(* PLC project binary_encoder, Dassault Systèmes ControlBuild 2024x *)
(* stored: creationDateTime 2023-10-03T11:12:52-01:00 *)

(* This module simulates the behaviour of a binary encoder *)
FUNCTION_BLOCK equipment_library.binary_encoder
  VAR_INPUT
    binaryInput : DINT := 0;
    encoderFreezing : BOOL := false;
  END_VAR
  VAR_OUTPUT
    bit00 : BOOL := false;
    bit01 : BOOL := false;
    bit02 : BOOL := false;
    bit03 : BOOL := false;
    bit04 : BOOL := false;
    bit05 : BOOL := false;
    bit06 : BOOL := false;
    bit07 : BOOL := false;
    bit08 : BOOL := false;
    bit09 : BOOL := false;
    bit10 : BOOL := false;
    bit11 : BOOL := false;
    bit12 : BOOL := false;
    bit13 : BOOL := false;
    bit14 : BOOL := false;
    bit15 : BOOL := false;
    bit16 : BOOL := false;
    wordOutput : DINT := 0;
  END_VAR
  VAR
    inputValue : DINT := 0;
    parity : BOOL := false;
  END_VAR
  VAR CONSTANT
    evenParity : BOOL := false;
    oddParity : BOOL := true;
  END_VAR
  VAR
    d_presetting : BOOL := false;
    v_d_presetting : DINT := 0;
  END_VAR


ACTION C_source_code:
/* ----------------------------------------------------------------	*/
/* Type : Model of Operative Behaviour					*/
/* Category :  Sensors							*/
/* Author : Dassault Systemes						*/
/* Update date : June 2018							*/
/* ----------------------------------------------------------------	*/
/* This module simulates the behaviour 					*/
/* of a binary encoder.							*/
/* The whole value is encoded on 15 bits					*/
/*	the 16th bit is the parity bit. 					*/
/* ----------------------------------------------------------------	*/

/* ----------------------------------------------------------------	*/
/* Treatment of presetting fault						*/
/* ----------------------------------------------------------------	*/
if (d_presetting) inputValue = v_d_presetting;
else inputValue = binaryInput;


/* ----------------------------------------------------------------	*/
/* Encoder management							*/
/* ----------------------------------------------------------------	*/
if (!encoderFreezing) {
	bit00 = 0;
	bit01 = 0;
	bit02 = 0;
	bit03 = 0;
	bit04 = 0;
	bit05 = 0;
	bit06 = 0;
	bit07 = 0;
	bit08 = 0;
	bit09 = 0;
	bit10 = 0;
	bit11 = 0;
	bit12 = 0;
	bit13 = 0;
	bit14 = 0;
	bit15 = 0;

	if ((inputValue & 1)>0) bit00 = 1;
	if ((inputValue & 2)>0) bit01 = 1;
	if ((inputValue & 4)>0) bit02 = 1;
	if ((inputValue & 8)>0) bit03 = 1;
	if ((inputValue & 16)>0) bit04 = 1;
	if ((inputValue & 32)>0) bit05 = 1;
	if ((inputValue & 64)>0) bit06 = 1;
	if ((inputValue & 128)>0) bit07 = 1;
	if ((inputValue & 256)>0) bit08 = 1;
	if ((inputValue & 512)>0) bit09 = 1;
	if ((inputValue & 1024)>0) bit10 = 1;
	if ((inputValue & 2048)>0) bit11 = 1;
	if ((inputValue & 4096)>0) bit12 = 1;
	if ((inputValue & 8192)>0) bit13 = 1;
	if ((inputValue & 16384)>0) bit14 = 1;
	if ((inputValue & 32768)>0) bit15 = 1;

	/* -----------------------------------------------------------------------------------------------------------	*/
	/* 	Calcul de la parity : Si parity = 0 => parity paire		*/
	/* -----------------------------------------------------------------------------------------------------------	*/
	parity =((((((((((((((bit00 ^ bit01) ^ bit02) ^ bit03) ^ bit04) ^ bit05) ^ bit06) ^ bit07) ^ bit08)
			 ^ bit09) ^ bit10) ^ bit11) ^ bit12) ^ bit13) ^ bit14);

	if (evenParity && !oddParity) bit15 = parity;
	else if(!evenParity && oddParity) bit15 = !parity;

	/* -----------------------------------------------------------------------------------------------------------	*/
	/*	Traitement sortie sur mot						*/
	/* -----------------------------------------------------------------------------------------------------------	*/
	wordOutput = 0;
	if (bit00)  wordOutput = wordOutput + 1;
	if (bit01)  wordOutput = wordOutput + 2;
	if (bit02)  wordOutput = wordOutput + 4;
	if (bit03)  wordOutput = wordOutput + 8;
	if (bit04)  wordOutput = wordOutput + 16;
	if (bit05)  wordOutput = wordOutput + 32;
	if (bit06)  wordOutput = wordOutput + 64;
	if (bit07)  wordOutput = wordOutput + 128;
	if (bit08)  wordOutput = wordOutput + 256;
	if (bit09)  wordOutput = wordOutput + 512;
	if (bit10)  wordOutput = wordOutput + 1024;
	if (bit11)  wordOutput = wordOutput + 2048;
	if (bit12)  wordOutput = wordOutput + 4096;
	if (bit13)  wordOutput = wordOutput + 8192;
	if (bit14)  wordOutput = wordOutput + 16384;
	if (bit15)  wordOutput = wordOutput + 32768;
}
END_ACTION
END_FUNCTION_BLOCK
